TYPE GridPoint :
STRUCT
	x, y : INT;
END_STRUCT
END_TYPE

(* stored: Version 1.1.0.1, ProductVersion 3.1.4024.11
   DUT GridPoint: Id {200bbd50-9c3c-49d3-929b-1a300f154865} *)
